TYPE RobotJob : STRUCT
		jobNumber : INT;
END_STRUCT
END_TYPE

(* stored: Version 1.1.0.1, ProductVersion 3.1.4024.11
   DUT RobotJob: Id {75db9127-bb31-47ac-9783-5f3b759e71e0} *)
